FUNCTION HasExtensionNamespace : BOOL
VAR_INPUT
	Symbol : T_MAXSTRING;
END_VAR
VAR
	splitNamespace : t_MAXSTRING;
    splitSymbol : T_MAXSTRING;
END_VAR

HasExtensionNamespace := FindAndSplitChar( 
	sSeparatorChar := '.',  
	pSrcString := ADR(Symbol),                                  
	pLeftString := ADR(splitNamespace),   
	nLeftSize := SIZEOF(splitNamespace),                                  
	pRightString := ADR(splitSymbol), 
	nRightSize := SIZEOF(splitSymbol),                                
	bSearchFromRight := FALSE 
);

END_FUNCTION

(* stored: Version 1.1.0.1, ProductVersion 3.1.4024.12
   POU HasExtensionNamespace: Id {72ed1bbb-a749-0ec4-31e0-d56410b294d3}, SpecialFunc None *)
